FUNCTION_BLOCK SetEnabledProcess EXTENDS BaseProcess
VAR_INPUT
	///Arguments to be set, before writing do_request TRUE
	{attribute 'OPC.UA.DA' := '1'}
	set: SetEnabledProcessArgs;
END_VAR
VAR_OUTPUT
	///Arguments in use by the process, if do_request was accepted
	{attribute 'OPC.UA.DA' := '1'}
	{attribute 'OPC.UA.DA.Access' := '1'}
	get: SetEnabledProcessArgs;
END_VAR
VAR_IN_OUT
END_VAR
VAR
END_VAR

IF do_request THEN
    do_request_result := request( enabled := set.enabled );
    do_request := FALSE;
END_IF;
SUPER^();

{attribute 'TcRpcEnable' := '1'}
METHOD start
VAR_INPUT
	///True to enable, false to disable
	enabled: BOOL;
END_VAR
VAR_OUTPUT
END_VAR
VAR_IN_OUT
END_VAR
VAR
END_VAR
THIS^.get.enabled := enabled;
THIS^.statuses.busyStatus( isBusy := TRUE );
THIS^.statuses.healthStatus( isGood := TRUE );
END_METHOD

{attribute 'TcRpcEnable' := '1'}
METHOD request : RequestResults
VAR_INPUT
	///True to enable, false to disable
	enabled: BOOL;
END_VAR
VAR_OUTPUT
END_VAR
VAR_IN_OUT
END_VAR
VAR
END_VAR
IF THIS^.statuses.enabledStatus.enabled THEN
    THIS^.start( enabled := enabled );
    request := RequestResults.ACCEPTED;
ELSE
    request := RequestResults.REJECTED;
END_IF;
END_METHOD

END_FUNCTION_BLOCK

(* stored: Version 1.1.0.1, ProductVersion 3.1.4019.2
   POU SetEnabledProcess: Id {e5be4e0c-fab7-42fe-bb30-c72a18bbcf37}, SpecialFunc None
   Method start: Id {44ed64ad-8bf2-4b77-9cd4-909f3275515f}
   Method request: Id {d7c6b44a-4f23-4ec5-92bc-b64bd9c92852} *)
